INTERFACE PUBLIC I_HomingBuilder EXTENDS __System.IQueryInterface

METHOD BuildForceCalibrationCommand : HomingCommand
END_METHOD

METHOD BuildResetCalibrationCommand : HomingCommand
END_METHOD

METHOD Position : I_PositioningHomingBuilder
VAR_INPUT
	value : LREAL;
END_VAR
END_METHOD

END_INTERFACE

(* stored: Version 1.1.0.1, ProductVersion 3.1.4026.13
   Itf I_HomingBuilder: Id {1502ebfb-6262-0c79-05bd-2fcc0e8b4561}
   Method BuildForceCalibrationCommand: Id {ee6c6235-136e-0786-13e2-899bf3e8c5f3}
   Method BuildResetCalibrationCommand: Id {2866cf16-5cd8-05fa-19c4-e1f7c57f03c4}
   Method Position: Id {f1f9add0-954b-0697-2815-fe57829c420f} *)
